TYPE ST_SettingsLiftingTransport :
STRUCT
	//Param file
	bAutoRecoveryToIdle : BOOL;	//Auto recovery to Idle-position in case of failure e.g.: (un)locking trolley failed
	tTrolleyUnLockCheckMinTime : TIME; //Trolley (Un)Locked check minimal time
	tTrolleyUnLockCheckMaxTime : TIME; //Trolley (Un)Locked check maximal time (time out)
	tTrolleyAtCabinCheckMinTime : TIME; //Trolley at cabin position check minimal time
	tTrolleyAtCabinCheckMaxTime : TIME; //Trolley at cabin position check maximal time (time out)
	bWaitForNextStep : BOOL; //Wait for next button to be pressed before starting new positioning step
	
	//Init Config
	stSettingsServoLift : ST_SettingsServo;
	arr_stLiftPositioningProfile : ARRAY[0..10] OF ST_PositioningProfile;
	
	stSettingsServoTransport : ST_SettingsServo;
	arr_stTransportPositioningProfile : ARRAY[0..5] OF ST_PositioningProfile;
	
	END_STRUCT
END_TYPE

(* stored: Version 1.1.0.1, ProductVersion 3.1.4024.12
   DUT ST_SettingsLiftingTransport: Id {cad671c8-daf9-4539-9908-38693c7e494e} *)
